# B&R Automation Studio project Analog
Automation Studio 4.9

## Configuration Config1

CPU X20CP0484, AutomationRuntime 6.5.1, Build 11.3.0, Vc 6.0.0

### Task classes (Cpu.sw)
```
Cyclic#4 (cycle 100000 us, tolerance 100000 us):
  Program <- Program.prg
Libraries: AsIecCon, runtime
```

### Hardware
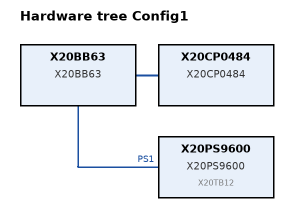
```
X20BB63 : X20BB63 v1.1.0.0
X20CP0484 : X20CP0484 v1.8.1.0  [SL -> X20BB63.SL1]
  Connector IF2:
    ActivateDevice = 1
  ConfigurationID = Analog_Config1
  Simulation = 1
  TimerDeviceType = SWIOTIMER
  Cyclic1Duration = 10000
  Cyclic1Tolerance = 10000
  Cyclic2Duration = 20000
  Cyclic2Tolerance = 20000
  Cyclic3Duration = 50000
  Cyclic3Tolerance = 50000
  Cyclic4Duration = 100000
  Cyclic4Tolerance = 100000
  Cyclic5Duration = 200000
  Cyclic5Tolerance = 200000
  Cyclic6Duration = 500000
  Cyclic6Tolerance = 500000
  Cyclic7Duration = 1000000
  Cyclic7Tolerance = 1000000
  Cyclic8Duration = 10000
  Cyclic8Tolerance = 30000000
  FileDevice1
  FileDeviceName1 = USER
  FileDevicePath1 = USER_PATH
X20PS9600 : X20PS9600 v1.6.2.0  [PS -> X20BB63.PS1; SS1 -> X20TB12.SS]
X20TB12 : X20TB12 v1.0.0.0
```

## Logical view

### Program Logical/Program (IEC)

#### Main.st - Init, cyclic, exit code
```iecst
PROGRAM _INIT
	(* Insert code here *)
	analog1Config.HSV := 20;
	analog1Config.LSV := 0;
	analog1Config.SensorType := Pressure;
	analog1Config.Signal:= voltage0_10;
END_PROGRAM

PROGRAM _CYCLIC
	(* Insert code here *)
	fb_Analog(Config := analog1Config,RAW := auxTest);
	analog := fb_Analog.AnalogOUT;

	fb_Analog_2.Config.HSV := 100;
	fb_Analog_2.RAW := auxTest;
	fb_Analog_2.Config.LSV := 0;
	fb_Analog_2();
	analog_2 := fb_Analog_2.AnalogOUT;

END_PROGRAM

PROGRAM _EXIT
	(* Insert code here *)

END_PROGRAM
```

#### Types.typ - Local data types
```iecst
TYPE
	SensorsType :
		(
		Pressure,
		Temp,
		Angle
		);
	SignalType :
		(
		voltage0_10,
		milliamps0_20,
		milliamps4_20
		);
	Configuration : 	STRUCT
		LSV : REAL;
		HSV : REAL;
		SensorType : SensorsType;
		Signal : SignalType;
	END_STRUCT;
END_TYPE
```

#### Variables.var - Local variables
```iecst
VAR
	fb_Analog : Name;
	auxTest : INT;
	analog : REAL;
	fb_Analog_2 : Name;
	analog_2 : REAL;
	analog1Config : Configuration;
END_VAR
```

#### LocalFunctions.fun
```iecst
{REDUND_ERROR} FUNCTION_BLOCK Name (*TODO: Add your comment here*) (*$GROUP=User,$CAT=User,$GROUPICON=User.png,$CATICON=User.png*)
	VAR
		New_Member : USINT;
	END_VAR
	VAR_INPUT
		test : {REDUND_UNREPLICABLE} BOOL;
	END_VAR
END_FUNCTION_BLOCK
```

#### Name.st
```iecst
(* TODO: Add your comment here *)
FUNCTION_BLOCK Name

	AnalogOUT := INT_TO_REAL( REAL_TO_INT(AnalogOUT*100))/100;(*Zaokrąglenie wyjscia analogowego*)
	//AnalogOutSignal := Scale(0,Normalize(0,RAW,32768),20);

	AnalogOut10 := REAL_TO_INT(AnalogOUT*10);
	AnalogOut100 := REAL_TO_INT(AnalogOUT*100);
	CASE Config.Signal OF
		voltage0_10:
			AnalogOutSignal := INT_TO_REAL( REAL_TO_INT(Scale(0,Normalize(0,RAW,32768),10)*100)/100);
		milliamps0_20:
			AnalogOutSignal := INT_TO_REAL( REAL_TO_INT(Scale(0,Normalize(0,RAW,32768),20)*100)/100);
		milliamps4_20:
			AnalogOutSignal := INT_TO_REAL( REAL_TO_INT(Scale(4,Normalize(0,RAW,32768),20)*100)/100);

	END_CASE;
	CASE Config.SensorType OF
		Pressure:
			AnalogOUT := Scale(Config.LSV, Normalize(0,RAW,32768),Config.HSV);
		Temp:
			AnalogOUT := Scale(Config.LSV, Normalize(0,RAW,32768),Config.HSV);
			AnalogOutKelvin := AnalogOUT + 273.15 ;
		Angle:
			AnalogOUT := Scale(0, Normalize(0,RAW,32768),360);

	END_CASE;

	IF Config.HSV = 0 THEN
		Error := TRUE ;
	END_IF
	IF Error THEN
		AnalogOUT := 0;
		AnalogOut10 := 0;
		AnalogOut100 := 0;
		AnalogOutSignal := 0;
		AnalogOutKelvin := 0;
	END_IF

END_FUNCTION_BLOCK
```

#### Scale.st
```iecst
(* TODO: Add your comment here *)
FUNCTION Scale
	Scale :=  (Value *(Maximum-Minimum)) + Minimum;
END_FUNCTION
```

#### Normalize.st
```iecst
(* TODO: Add your comment here *)
FUNCTION Normalize
	Normalize :=(Value - Minimum)/(Maximum - Minimum);
END_FUNCTION
```
